INTERFACE I_Pizza

METHOD GetPrice : LREAL
VAR_INPUT
END_VAR
END_METHOD

END_INTERFACE

(* stored: Version 1.1.0.1, ProductVersion 3.1.4022.12
   Itf I_Pizza: Id {94ba4d5f-9647-4942-b8c6-1fc8ff98a453}
   Method GetPrice: Id {33df6340-b453-4bcc-8f4a-647dd0046888} *)
